FUNCTION_BLOCK fb_modeController
VAR_INPUT
END_VAR
VAR_OUTPUT
END_VAR
VAR
	SFCInit : BOOL;
	trn_autoRun: BOOL;
	fbi_manual: fb_manual;
	fbi_auto: fb_auto;
	fbi_paramInit: fb_paramInit;	
	trn_autoDone: BOOL;
	var_process: INT;
	fbi_delayTimer0: TON;
	fbi_delayTimer1: TON;
	fbi_delayTimer2: TON;
	fbi_delayTimer3: TON;
	MC_ResetX: MC_Reset;
	MC_ResetY: MC_Reset;
	MC_ResetZ: MC_Reset;
	trn_SaftyUnitResetDone: BOOL;
	resetDelay: TON;
	MC_ResetR: MC_Reset;
	MC_Stop_x: MC_Stop;
	MC_Stop_y: MC_Stop;
	MC_Stop_z: MC_Stop;
	MC_Stop_r: MC_Stop;
	fbi_delayTimer4: TON;
	fbi_timer: TON;
END_VAR
VAR_STAT
	
END_VAR

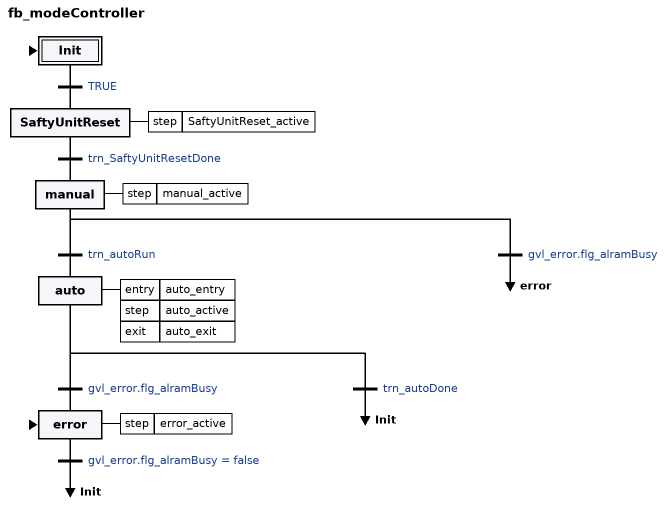
INITIAL_STEP Init:
END_STEP
TRANSITION FROM Init TO SaftyUnitReset
    := TRUE;
END_TRANSITION
STEP SaftyUnitReset:
    SaftyUnitReset_active(N);  // step action
END_STEP
TRANSITION FROM SaftyUnitReset TO manual
    := trn_SaftyUnitResetDone;
END_TRANSITION
STEP manual:
    manual_active(N);  // step action
END_STEP
TRANSITION FROM manual TO auto
    := trn_autoRun;
END_TRANSITION
TRANSITION FROM manual TO error
    := gvl_error.flg_alramBusy;
END_TRANSITION
STEP auto:
    auto_entry(P1);  // entry action
    auto_active(N);  // step action
    auto_exit(P0);  // exit action
END_STEP
TRANSITION FROM auto TO error
    := gvl_error.flg_alramBusy;
END_TRANSITION
TRANSITION FROM auto TO Init
    := trn_autoDone;
END_TRANSITION
STEP error:
    error_active(N);  // step action
END_STEP
TRANSITION FROM error TO Init
    := gvl_error.flg_alramBusy = false;
END_TRANSITION

ACTION auto_active:
IF auto._x AND auto.x = FALSE THEN
	gvl_io.flg_signalTowerGreen := TRUE;
	gvl_io.flg_signalTowerYellow := FALSE;
	gvl_io.flg_signalTowerRed := FALSE;
	trn_autoDone := FALSE;
	THIS^.fbi_auto.p_Init := TRUE;
	THIS^.fbi_auto();
	gvl_auto.requirementToPickUpLens := FALSE;
	gvl_visu.flg_btn_autoModeStop := FALSE;
	gvl_auto.autoModeStoped := FALSE;
	gvl_auto.autoModeStop := FALSE;
	
	gvl_axis.ref_x.Velocity 	:= gvl_param.var_productInfo[gvl_param.var_currentProductID].autoVels.x.vel;
	gvl_axis.ref_x.Acceleration	:= gvl_param.var_productInfo[gvl_param.var_currentProductID].autoVels.x.acc;
	gvl_axis.ref_x.Deceleration	:= gvl_param.var_productInfo[gvl_param.var_currentProductID].autoVels.x.dcc;
	gvl_axis.ref_y.Velocity		:= gvl_param.var_productInfo[gvl_param.var_currentProductID].autoVels.y.vel;
	gvl_axis.ref_y.Acceleration	:= gvl_param.var_productInfo[gvl_param.var_currentProductID].autoVels.y.acc;
	gvl_axis.ref_y.Deceleration	:= gvl_param.var_productInfo[gvl_param.var_currentProductID].autoVels.y.dcc;
	gvl_axis.ref_z.Velocity		:= gvl_param.var_productInfo[gvl_param.var_currentProductID].autoVels.z.vel;
	gvl_axis.ref_z.Acceleration	:= gvl_param.var_productInfo[gvl_param.var_currentProductID].autoVels.z.acc;
	gvl_axis.ref_z.Deceleration	:= gvl_param.var_productInfo[gvl_param.var_currentProductID].autoVels.z.dcc;
	gvl_axis.ref_r.Velocity		:= gvl_gm.var_buf_autoVel;
	gvl_axis.ref_r.Acceleration	:= gvl_gm.var_buf_autoAcc;
	gvl_axis.ref_r.Deceleration	:= gvl_gm.var_buf_autoDec;
	gvl_param.var_currentMode := eP_programMode.auto;
ELSIF auto._x AND auto.x THEN
	gvl_visu.flg_btn_invalidBuzzer := FALSE;
	THIS^.fbi_auto.p_Init := FALSE;
	THIS^.fbi_auto();
	IF gvl_visu.flg_btn_autoModeStop THEN
		gvl_auto.autoModeStop := TRUE;
	END_IF
	IF gvl_auto.autoModeStoped THEN
		trn_autoDone := TRUE;
	END_IF
END_IF
END_ACTION

ACTION auto_entry:
gvl_auto.requirementToPickUpLens := FALSE;
gvl_auto.autoModeStoped := FALSE;
gvl_auto.autoModeStop := FALSE;
gvl_auto.flg_gm_measurementClosed := FALSE;
gvl_auto.flg_gm_transportClosed := FALSE;
gvl_auto.flg_transportClosed := false;
END_ACTION

ACTION auto_exit:
gvl_auto.requirementToPickUpLens := FALSE;
gvl_auto.autoModeStoped := FALSE;
gvl_auto.autoModeStop := FALSE;
gvl_auto.flg_gm_measurementClosed := FALSE;
gvl_auto.flg_gm_transportClosed := FALSE;
gvl_auto.flg_transportClosed := FALSE;
gvl_io.flg_requestLens := FALSE;
gvl_auto.flg_axisIsPcikingUp := FALSE;
gvl_auto.flg_gm_eleIsDown := FALSE;
gvl_visu.flg_btn_sample := FALSE;
gvl_gm.var_incjetInfo.flg_denyStamp := FALSE;
END_ACTION

ACTION error_active:
IF error._x AND error.x = FALSE THEN
	gvl_io.flg_signalTowerGreen := FALSE;
	gvl_io.flg_signalTowerYellow := FALSE;
	gvl_axis.fbi_motionControler.p_Init := TRUE;
	gvl_param.var_currentMode := eP_programMode.error;
	fbi_paramInit.in_flg_run := FALSE;
	fbi_delayTimer0.in := FALSE;
	fbi_delayTimer1.IN := FALSE;
	fbi_delayTimer2.IN := FALSE;
	fbi_delayTimer3.IN := FALSE;
	fbi_delayTimer4.IN := FALSE;
	var_process := 0;
ELSIF error._x AND error.x THEN
	CASE var_process OF
		0:
			MC_Stop_x.Execute := TRUE;
			MC_Stop_y.Execute := TRUE;
			MC_Stop_z.Execute := TRUE;
			IF gvl_visu.flg_btn_usingMeasurementSystem THEN
				MC_Stop_r.Execute := TRUE;
			END_IF
			var_process := 1;
		1:
			MC_Stop_x.Execute := FALSE;
			MC_Stop_y.Execute := FALSE;
			MC_Stop_z.Execute := FALSE;	
			MC_Stop_r.Execute := FALSE;	
			IF gvl_error.flg_reset THEN
				var_process := 2;
			END_IF
		2:
			gvl_io.var_gateMeasurementReset := 0;
			gvl_error.flg_vacuum := FALSE;
			gvl_error.flg_fiberSens := FALSE;
			gvl_error.flg_gm_fiberSens := FALSE;
			gvl_error.flg_incjet := FALSE;
			gvl_error.flg_sample_windown_error:= FALSE;
			gvl_axis.fbi_motionControler.p_Init := FALSE;
			fbi_paramInit.in_flg_run := TRUE;
			gvl_io.var_gateMeasurementReset := 1;
			IF fbi_paramInit.out_flg_done THEN
				fbi_paramInit.in_flg_run := FALSE;
				gvl_visu.var_msg:="";
				var_process := 3;
			END_IF
		3:
			fbi_delayTimer0.IN := TRUE;
			gvl_io.flg_saftyUnitReset := TRUE;
			IF fbi_delayTimer0.Q THEN
				gvl_io.flg_saftyUnitReset := FALSE;
				var_process := 7;
			END_IF
//		4:
//			gvl_elecylinder.fbi_gm_axisTransport.in_flg_run := FALSE;
//			gvl_elecylinder.fbi_gm_axisPickUp.in_flg_run := FALSE;
//			var_process := 5;
//		5:
//			gvl_elecylinder.fbi_gm_axisTransport.in_var_moveMode := eP_eleMoveMode.eleA;
//			gvl_elecylinder.fbi_gm_axisPickUp.in_var_moveMode := eP_eleMoveMode.eleA;
//			gvl_elecylinder.fbi_gm_axisTransport.in_flg_run := TRUE;
//			gvl_elecylinder.fbi_gm_axisPickUp.in_flg_run := TRUE;
//			var_process := 6;
//		6:
//			IF gvl_elecylinder.fbi_gm_axisTransport.out_flg_Done AND gvl_elecylinder.fbi_gm_axisPickUp.out_flg_Done THEN
//				gvl_elecylinder.fbi_gm_axisTransport.in_flg_run := FALSE;
//				gvl_elecylinder.fbi_gm_axisPickUp.in_flg_run := FALSE;
//				var_process := 7;
//			END_IF
		7:
			gvl_io.flg_saftyUnitReset := FALSE;
			MC_ResetX.Execute := TRUE;
			MC_ResetY.Execute := TRUE;
			MC_ResetZ.Execute := TRUE;
			MC_ResetR.Execute := TRUE;
			gvl_elecylinder.ref_axis_transport.output.out_flg_reset := TRUE;
			gvl_elecylinder.ref_axis_sample.output.out_flg_reset := TRUE;
			gvl_elecylinder.ref_axis_trayChange.output.out_flg_reset := TRUE;
			gvl_elecylinder.ref_axis_rotary.output.out_flg_reset := TRUE;
			var_process := 8;
		8:
			MC_ResetX.Execute := FALSE;
			MC_ResetY.Execute := FALSE;
			MC_ResetZ.Execute := FALSE;
			MC_ResetR.Execute := FALSE;
			gvl_elecylinder.ref_axis_transport.output.out_flg_reset := FALSE;
			gvl_elecylinder.ref_axis_sample.output.out_flg_reset := FALSE;
			gvl_elecylinder.ref_axis_trayChange.output.out_flg_reset := FALSE;
			gvl_elecylinder.ref_axis_rotary.output.out_flg_reset := FALSE;
			fbi_delayTimer4.IN := TRUE;
			(*
			IF fbi_delayTimer4.Q THEN
				var_process := 6;
			END_IF
			*)
			IF gvl_io.in_wire_saftyUnitState THEN
				var_process := 9;
			ELSIF fbi_delayTimer4.Q THEN
				var_process := 9;
			END_IF
		9:	
			gvl_error.flg_resetEventFlg := TRUE;
			fbi_delayTimer1.IN := TRUE;
			IF fbi_delayTimer1.Q THEN
				var_process := 10;
			END_IF
		10:
			gvl_error.flg_eventDisplayRest := TRUE;
			fbi_delayTimer2.IN := TRUE;
			IF fbi_delayTimer2.Q THEN
				var_process := 11;
			END_IF
		11:
			fbi_delayTimer3.IN := TRUE;
			gvl_error.flg_ararmLevelRest := TRUE;
			IF fbi_delayTimer3.Q  THEN
				var_process := 12;
			END_IF
		12:
			gvl_error.flg_resetEventFlg := FALSE;
			gvl_error.flg_eventDisplayRest := FALSE;
			gvl_error.flg_ararmLevelRest := FALSE;
			gvl_error.flg_alramBusy := FALSE;
						
	END_CASE
END_IF
MC_ResetX(
	Axis:= gvl_axis.axisX , 
	Execute:= , 
	Done=> , 
	Busy=> , 
	Error=> , 
	ErrorID=> );
MC_ResetY(
	Axis:= gvl_axis.axisY , 
	Execute:= , 
	Done=> , 
	Busy=> , 
	Error=> , 
	ErrorID=> );
MC_ResetZ(
	Axis:= gvl_axis.axisZ , 
	Execute:= , 
	Done=> , 
	Busy=> , 
	Error=> , 
	ErrorID=> );
MC_ResetR(
	Axis:= gvl_axis.axisR , 
	Execute:= , 
	Done=> , 
	Busy=> , 
	Error=> , 
	ErrorID=> );
MC_Stop_x(
	Axis:= gvl_axis.axisX, 
	Execute:= , 
	Deceleration:= , 
	Jerk:= , 
	Options:= , 
	Done=> , 
	Busy=> , 
	Active=> , 
	CommandAborted=> , 
	Error=> , 
	ErrorID=> );
MC_Stop_y(
	Axis:= gvl_axis.axisY, 
	Execute:= , 
	Deceleration:= , 
	Jerk:= , 
	Options:= , 
	Done=> , 
	Busy=> , 
	Active=> , 
	CommandAborted=> , 
	Error=> , 
	ErrorID=> );
MC_Stop_z(
	Axis:= gvl_axis.axisZ, 
	Execute:= , 
	Deceleration:= , 
	Jerk:= , 
	Options:= , 
	Done=> , 
	Busy=> , 
	Active=> , 
	CommandAborted=> , 
	Error=> , 
	ErrorID=> );
MC_Stop_r(
	Axis:= gvl_axis.axisR, 
	Execute:= , 
	Deceleration:= , 
	Jerk:= , 
	Options:= , 
	Done=> , 
	Busy=> , 
	Active=> , 
	CommandAborted=> , 
	Error=> , 
	ErrorID=> );
	
	
fbi_delayTimer0(IN:= , PT:=T#500MS , Q=> , ET=> );
fbi_delayTimer1(IN:= , PT:=T#1000MS , Q=> , ET=> );
fbi_delayTimer2(IN:= , PT:=T#100MS , Q=> , ET=> );
fbi_delayTimer3(IN:= , PT:=T#100MS , Q=> , ET=> );
fbi_delayTimer4(IN:= , PT:=T#9000MS , Q=> , ET=> );
fbi_paramInit(in_flg_run:= , out_flg_done=> );
END_ACTION

ACTION manual_active:

IF manual._x AND manual.x = FALSE THEN
	gvl_io.flg_signalTowerGreen := FALSE;
	gvl_io.flg_signalTowerYellow := TRUE;
	gvl_io.flg_signalTowerRed := FALSE;
	gvl_visu.flg_btn_sample := FALSE;
	trn_autoRun := FALSE;
	gvl_visu.flg_btn_autoModeStart := FALSE;
	gvl_gm.var_incjetInfo.flg_denyStamp := FALSE;
	THIS^.fbi_manual();
	THIS^.fbi_manual.p_Init := TRUE;
ELSIF manual._x AND manual.x THEN
	THIS^.fbi_manual();
	THIS^.fbi_manual.p_Init := FALSE;
	gvl_auto.flg_transportClosed := FALSE;
	gvl_param.var_currentMode := eP_programMode.manual;
	gvl_io.flg_requestLens := FALSE;
	IF gvl_visu.flg_btn_autoModeStart THEN
		trn_autoRun := TRUE;
	END_IF
	gvl_param.var_productInfo[gvl_param.var_currentProductID].manaulVels.x.acc := 10000;
	gvl_param.var_productInfo[gvl_param.var_currentProductID].manaulVels.x.dcc := 10000;
	gvl_param.var_productInfo[gvl_param.var_currentProductID].manaulVels.y.acc := 10000;
	gvl_param.var_productInfo[gvl_param.var_currentProductID].manaulVels.y.dcc := 10000;
	gvl_param.var_productInfo[gvl_param.var_currentProductID].manaulVels.z.acc := 10000;
	gvl_param.var_productInfo[gvl_param.var_currentProductID].manaulVels.z.dcc := 10000;
 
	gvl_axis.ref_x.Velocity 	:= gvl_param.var_productInfo[gvl_param.var_currentProductID].manaulVels.x.vel;
	gvl_axis.ref_x.Acceleration := gvl_param.var_productInfo[gvl_param.var_currentProductID].manaulVels.x.acc;
	gvl_axis.ref_x.Deceleration := gvl_param.var_productInfo[gvl_param.var_currentProductID].manaulVels.x.dcc;
	gvl_axis.ref_y.Velocity 	:= gvl_param.var_productInfo[gvl_param.var_currentProductID].manaulVels.y.vel;
	gvl_axis.ref_y.Acceleration := gvl_param.var_productInfo[gvl_param.var_currentProductID].manaulVels.y.acc;
	gvl_axis.ref_y.Deceleration := gvl_param.var_productInfo[gvl_param.var_currentProductID].manaulVels.y.dcc;
	gvl_axis.ref_z.Velocity 	:= gvl_param.var_productInfo[gvl_param.var_currentProductID].manaulVels.z.vel;
	gvl_axis.ref_z.Acceleration := gvl_param.var_productInfo[gvl_param.var_currentProductID].manaulVels.z.acc;
	gvl_axis.ref_z.Deceleration := gvl_param.var_productInfo[gvl_param.var_currentProductID].manaulVels.z.dcc;
	gvl_axis.ref_r.Velocity 	:= gvl_gm.var_buf_manualVel;
END_IF
END_ACTION

PROPERTY p_init : bool
GET
p_init := THIS^.SFCInit;
END_GET
SET
THIS^.SFCInit := p_init;
END_SET
END_PROPERTY

ACTION SaftyUnitReset_active:
IF SaftyUnitReset._x AND SaftyUnitReset.x = FALSE THEN
	trn_SaftyUnitResetDone := FALSE;
	resetDelay.IN := FALSE;
	fbi_timer.IN := FALSE;
	gvl_io.flg_saftyUnitReset := TRUE;
	gvl_gm.var_incjetInfo.flg_denyStamp := FALSE;
ELSIF SaftyUnitReset._x AND SaftyUnitReset.x THEN
	resetDelay.IN := TRUE;
	fbi_timer.IN := True;
	IF resetDelay.Q THEN
		gvl_io.flg_saftyUnitReset := FALSE;
	END_IF
	
	IF gvl_io.flg_saftyUnitState THEN
		gvl_io.flg_saftyUnitReset := FALSE;
		trn_SaftyUnitResetDone := TRUE;
	ELSIF fbi_timer.Q THEN
		gvl_io.flg_saftyUnitReset := FALSE;
		trn_SaftyUnitResetDone := TRUE;
	END_IF
END_IF
resetDelay(IN:= , PT:=T#0.5S , Q=> , ET=> );
fbi_timer(IN:= , PT:=T#9S , Q=> , ET=> );
END_ACTION

END_FUNCTION_BLOCK

(* stored: Version 1.1.0.1, ProductVersion 3.1.4024.11
   POU fb_modeController: Id {35857279-3e84-4aaf-ab57-0c1e2bdefd85}, SpecialFunc None
   Action auto_active: Id {54b6a076-e02d-4cf1-9400-a90afa5e609d}
   Action auto_entry: Id {120b405a-a45d-4d72-9b88-f7c6c2708070}
   Action auto_exit: Id {d8a6f18d-17ca-46eb-b600-0fd32a86ea1d}
   Action error_active: Id {b98eb270-70d1-4d40-8b01-cf3d04788880}
   Action manual_active: Id {138234bc-e979-414c-a69b-939bfe534a52}
   Property p_init: Id {643651c5-dfb2-4f92-94eb-9507e978f203}
   Get Get: Id {8c766776-7e92-4d69-aaf6-31a179ae1315}
   Set Set: Id {42aaba73-160e-4db1-93db-5bd18e3b974a}
   Action SaftyUnitReset_active: Id {37337c83-ad80-4d5e-906f-1173f1500be2} *)
